(* IEC 61131-3 sources: RL_MAR/experiments/comparison/autoplc/results/qwen3.5-9b_20260511_180311/med_61, 1 file *)

(* ---- med_61_3.st ---- *)
FUNCTION_BLOCK FB_Sum
VAR_INPUT
    maxValue : INT;
END_VAR
VAR_OUTPUT
    wData : WORD;
END_VAR
VAR
    II : INT;
    tempSum : DINT;
END_VAR

    tempSum := 0;
    IF maxValue >= 0 THEN
        FOR II := 0 TO maxValue DO
            tempSum := tempSum + II;
        END_FOR;
    END_IF;
    wData := WORD(tempSum);
END_FUNCTION_BLOCK
